% RSLogix 500 project MM2-ATRIASIM_BAK038.RSS, saved by version 8.10.00.30 %
PROJECT "UNTITLED"    % processor: Bul.1763 MicroLogix 1100 Series B %

PROGRAM FILES
  LAD 2 "MAIN"  5 rungs
  LAD 3 "SAMPLECNT"  5 rungs
  LAD 4 "WATCHDOG"  8 rungs
  LAD 5 "SAMREG"  8 rungs  % Adding sample registratioon values to reg1 and 2 %
  LAD 6 "RESULTS"  8 rungs

DATA FILES
  O0 OUTPUT  4 elements
  I1 INPUT  6 elements
  S2 STATUS  66 elements
  B3 BINARY  1 elements
  T4 TIMER  2 elements
  C5 COUNTER  3 elements
  R6 CONTROL  1 elements
  N7 INTEGER  6 elements
  F8 FLOAT  8 elements

LADDER 2 "MAIN"
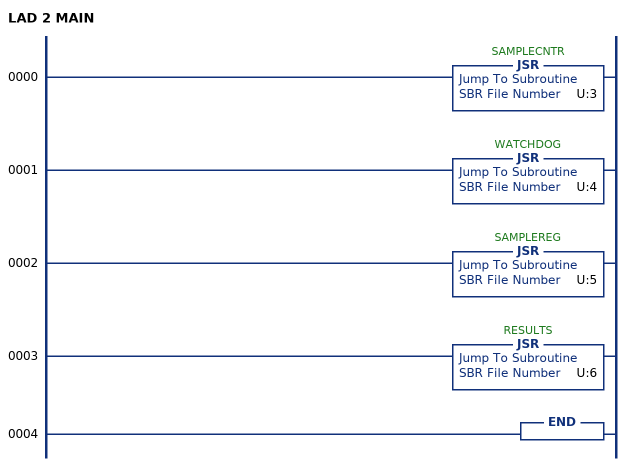
% Rung: 0 %
SOR JSR U:3 EOR
%   U:3  SAMPLECNTR %
% Rung: 1 %
SOR JSR U:4 EOR
%   U:4  WATCHDOG %
% Rung: 2 %
SOR JSR U:5 EOR
%   U:5  SAMPLEREG %
% Rung: 3 %
SOR JSR U:6 EOR
%   U:6  RESULTS %
% Rung: 4 %
SOR END EOR

LADDER 3 "SAMPLECNT"
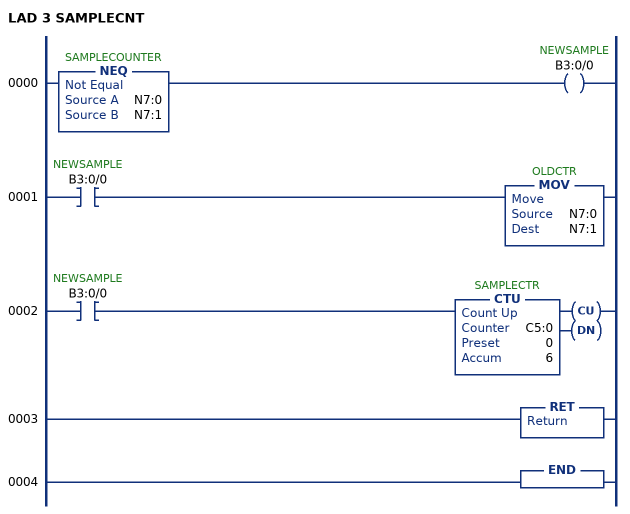
% Rung: 0 %
SOR NEQ N7:0 N7:1 OTE B3:0/0 EOR
%   N7:0  SAMPLECOUNTER %
%   N7:1  OLDCTR %
%   B3:0/0  NEWSAMPLE %
% Rung: 1 %
SOR XIC B3:0/0 MOV N7:0 N7:1 EOR
%   B3:0/0  NEWSAMPLE %
%   N7:0  SAMPLECOUNTER %
%   N7:1  OLDCTR %
% Rung: 2 %
SOR XIC B3:0/0 CTU C5:0 0 6 EOR
%   B3:0/0  NEWSAMPLE %
%   C5:0  SAMPLECTR %
% Rung: 3 %
SOR RET EOR
% Rung: 4 %
SOR END EOR

LADDER 4 "WATCHDOG"
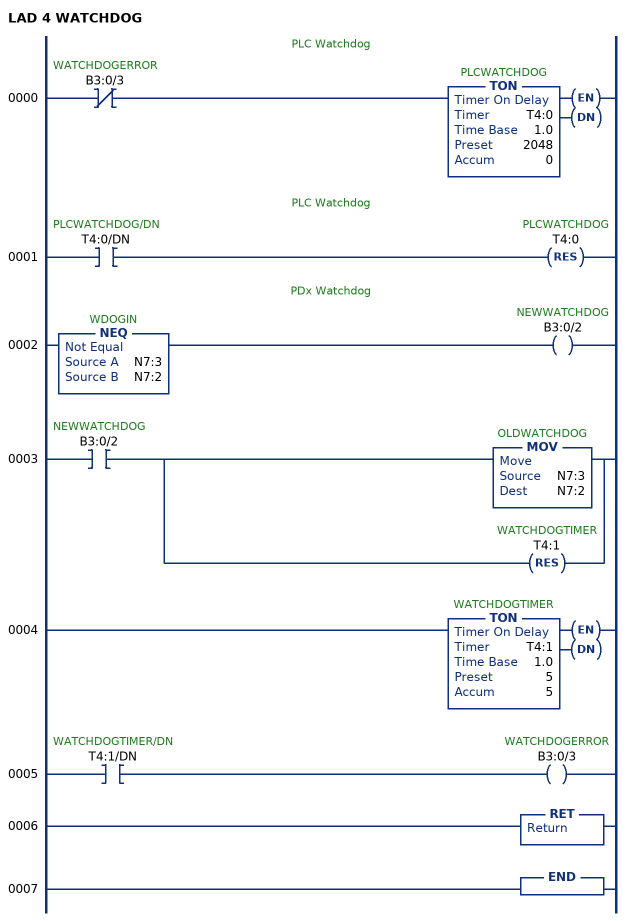
% Rung: 0 %
% PLC Watchdog %
SOR XIO B3:0/3 TON T4:0 1.0 2048 0 EOR
%   B3:0/3  WATCHDOGERROR %
%   T4:0  PLCWATCHDOG %
% Rung: 1 %
% PLC Watchdog %
SOR XIC T4:0/DN RES T4:0 EOR
%   T4:0  PLCWATCHDOG %
% Rung: 2 %
% PDx Watchdog %
SOR NEQ N7:3 N7:2 OTE B3:0/2 EOR
%   N7:3  WDOGIN %
%   N7:2  OLDWATCHDOG %
%   B3:0/2  NEWWATCHDOG %
% Rung: 3 %
SOR XIC B3:0/2 BST MOV N7:3 N7:2 NXB RES T4:1 BND EOR
%   B3:0/2  NEWWATCHDOG %
%   N7:3  WDOGIN %
%   N7:2  OLDWATCHDOG %
%   T4:1  WATCHDOGTIMER %
% Rung: 4 %
SOR TON T4:1 1.0 5 5 EOR
%   T4:1  WATCHDOGTIMER %
% Rung: 5 %
SOR XIC T4:1/DN OTE B3:0/3 EOR
%   T4:1  WATCHDOGTIMER %
%   B3:0/3  WATCHDOGERROR %
% Rung: 6 %
SOR RET EOR
% Rung: 7 %
SOR END EOR

LADDER 5 "SAMREG"    % Adding sample registratioon values to reg1 and 2 %
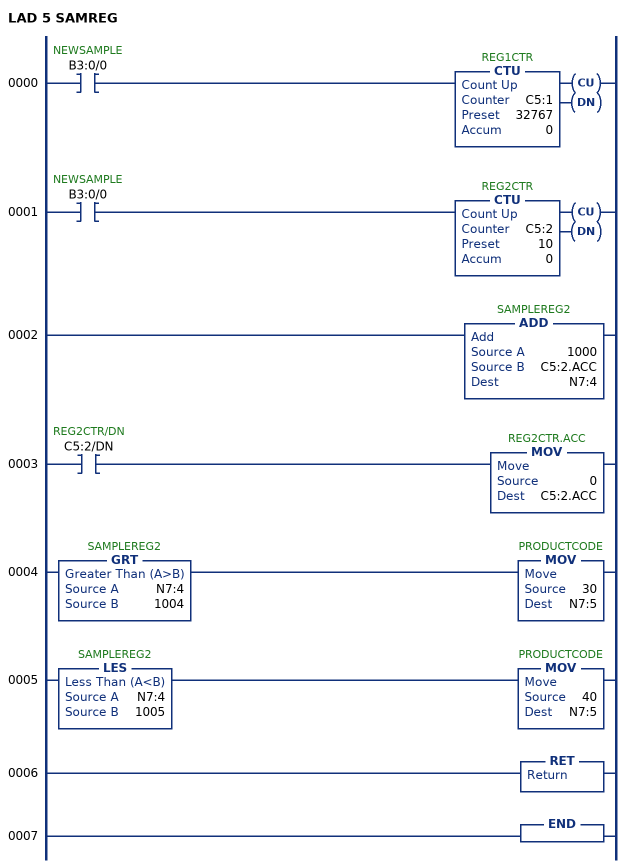
% Rung: 0 %
SOR XIC B3:0/0 CTU C5:1 32767 0 EOR
%   B3:0/0  NEWSAMPLE %
%   C5:1  REG1CTR %
% Rung: 1 %
SOR XIC B3:0/0 CTU C5:2 10 0 EOR
%   B3:0/0  NEWSAMPLE %
%   C5:2  REG2CTR %
% Rung: 2 %
SOR ADD 1000 C5:2.ACC N7:4 EOR
%   C5:2  REG2CTR %
%   N7:4  SAMPLEREG2 %
% Rung: 3 %
SOR XIC C5:2/DN MOV 0 C5:2.ACC EOR
%   C5:2  REG2CTR %
% Rung: 4 %
SOR GRT N7:4 1004 MOV 30 N7:5 EOR
%   N7:4  SAMPLEREG2 %
%   N7:5  PRODUCTCODE %
% Rung: 5 %
SOR LES N7:4 1005 MOV 40 N7:5 EOR
%   N7:4  SAMPLEREG2 %
%   N7:5  PRODUCTCODE %
% Rung: 6 %
SOR RET EOR
% Rung: 7 %
SOR END EOR

LADDER 6 "RESULTS"
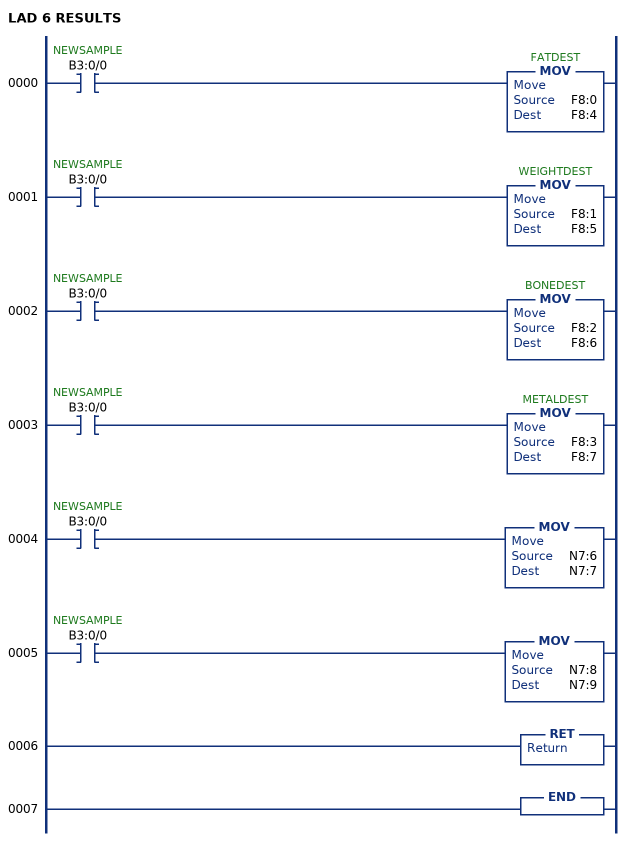
% Rung: 0 %
SOR XIC B3:0/0 MOV F8:0 F8:4 EOR
%   B3:0/0  NEWSAMPLE %
%   F8:0  FATRES %
%   F8:4  FATDEST %
% Rung: 1 %
SOR XIC B3:0/0 MOV F8:1 F8:5 EOR
%   B3:0/0  NEWSAMPLE %
%   F8:1  WEIGHTRES %
%   F8:5  WEIGHTDEST %
% Rung: 2 %
SOR XIC B3:0/0 MOV F8:2 F8:6 EOR
%   B3:0/0  NEWSAMPLE %
%   F8:2  BONERES %
%   F8:6  BONEDEST %
% Rung: 3 %
SOR XIC B3:0/0 MOV F8:3 F8:7 EOR
%   B3:0/0  NEWSAMPLE %
%   F8:3  METALRES %
%   F8:7  METALDEST %
% Rung: 4 %  % edit flag set %
SOR XIC B3:0/0 MOV N7:6 N7:7 EOR
%   B3:0/0  NEWSAMPLE %
%   N7:6  REF1RESULT %
% Rung: 5 %  % edit flag set %
SOR XIC B3:0/0 MOV N7:8 N7:9 EOR
%   B3:0/0  NEWSAMPLE %
%   N7:8  REF2RESULT %
% Rung: 6 %
SOR RET EOR
% Rung: 7 %
SOR END EOR

OTHER DOCUMENTED ADDRESSES
  B3:1/0  REF1RES
  B3:1/1  REF1DEST
  B3:1/2  REF2RES
  B3:1/3  REF2DEST

DATA TABLE (non-zero values as saved)
DATA T4
% .PRE .ACC %
% T4:0 % 2048 0
% T4:1 % 5 5
DATA C5
% .PRE .ACC %
% C5:0 % 0 6
% C5:1 % 32767 0
% C5:2 % 10 0
DATA N7
% N7:0 % 6 6 0 6 0 0
